INTERFACE I_Nci EXTENDS __System.IQueryInterface

PROPERTY _InternalNciPlcRef : REFERENCE TO NciPlc
GET
END_GET
END_PROPERTY

METHOD AddAxisToGroup
VAR_INPUT
	axis : I_Axis;
	index : UDINT;
	timeout : TIME;
	feedback : REFERENCE TO I_CommandFeedback;
END_VAR
END_METHOD

PROPERTY BlockNumber : UDINT
GET
END_GET
END_PROPERTY

METHOD BuildXYGroup
VAR_INPUT
	xAxis : I_Axis;
	yAxis : I_Axis;
	timeout : TIME;
	feedback : REFERENCE TO I_CommandFeedback;
END_VAR
END_METHOD

METHOD BuildXYZGroup
VAR_INPUT
	xAxis : I_Axis;
	yAxis : I_Axis;
	zAxis : I_Axis;
	timeout : TIME;
	feedback : REFERENCE TO I_CommandFeedback;
END_VAR
END_METHOD

PROPERTY ChannelId : UINT
GET
END_GET
END_PROPERTY

PROPERTY ChannelType : ChannelType
GET
END_GET
END_PROPERTY

PROPERTY ErrorId : UDINT
GET
END_GET
END_PROPERTY

METHOD GetGroupAxisIds : DWORD
VAR_IN_OUT
	axisIds : ARRAY[1..8] OF DWORD;
END_VAR
END_METHOD

METHOD GetOverride : LREAL
END_METHOD

PROPERTY GroupId : UDINT
GET
END_GET
END_PROPERTY

PROPERTY HandshakeableMFunction : INT
GET
END_GET
END_PROPERTY

PROPERTY HasError : BOOL
GET
END_GET
END_PROPERTY

PROPERTY HParam : DINT
GET
END_GET
END_PROPERTY

PROPERTY InterpreterState : UDINT
GET
END_GET
END_PROPERTY

PROPERTY IsEstop : BOOL
GET
END_GET
END_PROPERTY

METHOD IsFastMFunctionPresent : BOOL
VAR_INPUT
	functionNumber : INT;
END_VAR
END_METHOD

METHOD IsHandshakeableMFunctionPresent : BOOL
END_METHOD

METHOD ReadCyclicLRealParameter : LREAL
VAR_INPUT
	parameterNumber : UINT(1..4);
END_VAR
END_METHOD

METHOD ReadCyclicUdintParameter : UDINT
VAR_INPUT
	parameterNumber : UINT(1..4);
END_VAR
END_METHOD

METHOD ReleaseAxis
VAR_INPUT
	axis : I_Axis;
	timeout : TIME;
	feedback : REFERENCE TO I_CommandFeedback;
END_VAR
END_METHOD

METHOD ResetGroup
VAR_INPUT
	timeout : TIME;
	feedback : REFERENCE TO I_CommandFeedback;
END_VAR
END_METHOD

METHOD SetOverride : BOOL
VAR_INPUT
	value : LREAL;
END_VAR
END_METHOD

PROPERTY SetPathVelocity : LREAL
GET
END_GET
END_PROPERTY

PROPERTY SParam : UINT
GET
END_GET
END_PROPERTY

PROPERTY TParam : UINT
GET
END_GET
END_PROPERTY

END_INTERFACE

(* stored: Version 1.1.0.1, ProductVersion 3.1.4024.12
   Itf I_Nci: Id {570c7a38-6454-4db6-b650-0f44ec022371}
   Folder Configuration: Id {5ad4d588-929f-447c-8525-8985dad71904}
   Folder Internal Properties: Id {3072a58f-5ae4-4612-b701-7ca8877c1e3f}
   Folder Methods: Id {f77f3d23-fbba-47c6-b34e-0fc1790c53b1}
   Folder Properties: Id {eec006fe-b348-4f5c-9b54-a2b3ddd41320}
   Property _InternalNciPlcRef: Id {d01565a5-e48e-487e-b433-1877996b0254}
   Get Get: Id {25f1fee3-b16b-4515-bc31-f9d7680fde62}
   Method AddAxisToGroup: Id {444744cb-d6af-487e-b44f-ab8001ef7800}
   Property BlockNumber: Id {ab6139bd-d6d3-436d-b694-74030e428598}
   Get Get: Id {8f79da4b-eabd-4c36-9618-753a19affc2e}
   Method BuildXYGroup: Id {f30d86a5-c748-4f77-871f-3fc507770f31}
   Method BuildXYZGroup: Id {2d4d7752-4530-48c0-a358-46accab9a07e}
   Property ChannelId: Id {f15989cd-753a-4ccd-9228-d225dfdce9be}
   Get Get: Id {30379caa-df13-46f6-9cc8-06bd4d343fb2}
   Property ChannelType: Id {354f6c60-4c2f-4ceb-ac25-0186a007d5e1}
   Get Get: Id {3f34f902-86d2-451d-bf0e-5531bb8a0e15}
   Property ErrorId: Id {f2019ad9-5f70-4948-a532-822603389697}
   Get Get: Id {d6c11321-525b-40a8-a114-139ecfc1f5a0}
   Method GetGroupAxisIds: Id {1b582cbb-9aee-4bfd-88b0-60dc42111a4d}
   Method GetOverride: Id {fa575cad-dd0d-4950-b3f3-5fdb5a270672}
   Property GroupId: Id {83110107-eb25-4490-ad6f-fe3343ca6da0}
   Get Get: Id {e58a37f5-9c9b-4c1c-be80-cfca3f43ab84}
   Property HandshakeableMFunction: Id {9fa42292-8dfe-48e0-bc19-be0e4b20a074}
   Get Get: Id {7bc60249-32c2-4ee1-a1d9-8130a6436a45}
   Property HasError: Id {6b28ee11-6810-42f4-b700-5464e6b4d08c}
   Get Get: Id {91a6b5c4-a4ce-4eec-b198-a51a67579de3}
   Property HParam: Id {e0304bce-72e0-4242-8434-427da8eaf735}
   Get Get: Id {babcbf0b-2a6b-4018-8036-b2560b7a6cf9}
   Property InterpreterState: Id {16d1f98b-975c-457e-ad3d-d47eb4f286ed}
   Get Get: Id {670111f5-e362-481c-a1b4-9505fb30b375}
   Property IsEstop: Id {2ea9c9cd-8862-47d3-9854-f439692e71be}
   Get Get: Id {7fce7256-57cc-468e-9d7d-d4c717d43c51}
   Method IsFastMFunctionPresent: Id {9548f795-734f-45f8-b8ef-ac3e4a475645}
   Method IsHandshakeableMFunctionPresent: Id {cad43611-ae2e-456a-8678-ebf43a59a177}
   Method ReadCyclicLRealParameter: Id {55f674f9-875f-4540-a68f-669fc1f65c12}
   Method ReadCyclicUdintParameter: Id {f1e6773a-0eb4-4352-8846-40d6c9b46eee}
   Method ReleaseAxis: Id {fd96d428-8254-4e93-85a1-20c02f4c7001}
   Method ResetGroup: Id {8015ff9f-68f9-4bbb-8059-73c4c0a3a5b1}
   Method SetOverride: Id {98f77910-afe4-474f-bf0a-73893b3a8b09}
   Property SetPathVelocity: Id {4a78cc65-0702-4ead-bbdf-486a0a58b4b3}
   Get Get: Id {1e2c55d1-21c7-4426-ba53-7744843676fc}
   Property SParam: Id {3736a43a-d893-43a4-bcdf-ec95f485cecb}
   Get Get: Id {da2c3a18-680a-4c21-a6ce-528d9ef21b21}
   Property TParam: Id {937e6225-904b-40e8-9a66-10a39e340d28}
   Get Get: Id {74ed5602-1819-400f-a683-b07d88edd6ae} *)
